PROGRAM MAIN
VAR
	Test	:	BOOL;
END_VAR

IF GVL.MainPanel.StopPressed THEN
	
	GVL.MainPanel.StopLightOn();
	GVL.MainPanel.StartLightOff();

ELSIF GVL.MainPanel.StartPressed AND GVL.MainPanel.StopReleased THEN

	GVL.MainPanel.StopLightOff();
	GVL.MainPanel.StartLightOn();	

END_IF

END_PROGRAM

(* stored: Version 1.1.0.1, ProductVersion 3.1.4024.12
   POU MAIN: Id {8db4be02-5ee7-46ce-aa9f-b2ff94912b65}, SpecialFunc None *)
